// TwinCAT 3 PLC project PLC1
// Title: Projektnamn
// Company: Oaks AB
// ProgramVersion: 3.1.4023.0
// libraries:
//   OaksLibrary, * (OaksAB)
//   oaksModbusLibrary, * (Oaks AB)
//   Tc2_ModbusSrv, * (Beckhoff Automation GmbH)
//   Tc2_Standard, * (Beckhoff Automation GmbH)
//   Tc2_SUPS, * (Beckhoff Automation GmbH)
//   Tc2_System, * (Beckhoff Automation GmbH)
//   Tc2_Utilities, * (Beckhoff Automation GmbH)
//   Tc3_BA, * (Beckhoff Automation GmbH)
//   Tc3_Module, * (Beckhoff Automation GmbH)
// project tree:
//   GVLs/ IPadresser.TcGVL
//   / PlcTask.TcTTO
//   POUs/ImplicitChecks/ CheckBounds.TcPOU, CheckDivDInt.TcPOU, CheckDivLInt.TcPOU, CheckDivLReal.TcPOU, CheckDivReal.TcPOU, CheckLRangeSigned.TcPOU, CheckLRangeUnsigned.TcPOU, CheckRangeSigned.TcPOU, CheckRangeUnsigned.TcPOU
//   POUs/Lokala block/ fbDamperIndication_STL.TcPOU, fbfreezAlarm_markvarme.TcPOU, fbHeatPumpSr_StartStopDelay.TcPOU, fbReadAdsRealOutdoorMeantempWp_STL.TcPOU, fbTripleMotorControl_STL.TcPOU, fbTwinMotorControl_STL.TcPOU, fbTwinMotorHeatWoV.TcPOU
//   POUs/ MAIN.TcPOU
//   POUs/Övrigt/ AS101.TcPOU, KV1.TcPOU, S1.TcPOU, VVC1.TcPOU
// real-time tasks:
//   TASK PlcTask: cycle T#20ms, priority 20, ADS port 350
// I/O:
//   DEVICE Device 2 (CX-BK)
//     Box 1 (CX-BK)
// variable links:
//   PLC1/PLC1 Instance <-> Device 2 (CX-BK)/Box 1 (CX-BK)
//     PlcTask Inputs/AS101.AUT.V3 <-> Term 2 (KL1408)/Channel 6/Input
//     PlcTask Inputs/AS101.CBL.V3 <-> Term 2 (KL1408)/Channel 2/Input
//     PlcTask Inputs/AS101.FASBROTT.V3 <-> Term 2 (KL1408)/Channel 1/Input
//     PlcTask Inputs/AS101.JFB.V3 <-> Term 2 (KL1408)/Channel 4/Input
//     PlcTask Inputs/AS101.OSP.V3 <-> Term 2 (KL1408)/Channel 5/Input
//     PlcTask Inputs/AS101.RST.V <-> Term 2 (KL1408)/Channel 3/Input
//     PlcTask Inputs/AS101.SYSTEM.nKbusState <-> Inputs/State
//     PlcTask Inputs/KV1.PPA201_V <-> Term 5 (KL1408)/Channel 7/Input
//     PlcTask Inputs/S1.P11_QB_V3 <-> Term 2 (KL1408)/Channel 7/Input
//     PlcTask Inputs/S1.P12_QB_V3 <-> Term 4 (KL1408)/Channel 1/Input
//     PlcTask Inputs/S1.P13_QB_V3 <-> Term 4 (KL1408)/Channel 3/Input
//     PlcTask Inputs/S1.P14_QB_V3 <-> Term 4 (KL1408)/Channel 5/Input
//     PlcTask Inputs/S1.P15_QB_V3 <-> Term 4 (KL1408)/Channel 7/Input
//     PlcTask Inputs/S1.P16_QB_V3 <-> Term 5 (KL1408)/Channel 1/Input
//     PlcTask Inputs/S1.P17_QB_V3 <-> Term 5 (KL1408)/Channel 4/Input
//     PlcTask Inputs/S1.P11_V <-> Term 2 (KL1408)/Channel 8/Input
//     PlcTask Inputs/S1.P13_V <-> Term 4 (KL1408)/Channel 4/Input
//     PlcTask Inputs/S1.P15_V <-> Term 4 (KL1408)/Channel 8/Input
//     PlcTask Inputs/S1.P16_V <-> Term 5 (KL1408)/Channel 2/Input
//     PlcTask Inputs/S1.P17_V <-> Term 5 (KL1408)/Channel 5/Input
//     PlcTask Inputs/S1.P16_RC91_V <-> Term 5 (KL1408)/Channel 3/Input
//     PlcTask Inputs/S1.P17_RC91_V <-> Term 5 (KL1408)/Channel 6/Input
//     PlcTask Inputs/S1.ST1_P12_V <-> Term 4 (KL1408)/Channel 2/Input
//     PlcTask Inputs/S1.ST1_P14_V <-> Term 4 (KL1408)/Channel 6/Input
//     PlcTask Inputs/VVC1.GT420.iDataIn <-> Term 7 (KL3208-0010-4)/Channel 1/Data In
//     PlcTask Inputs/VVC1.GT420.usiState <-> Term 7 (KL3208-0010-4)/Channel 1/State
//     PlcTask Outputs/AS101.TCH1_bOutput <-> Term 3 (KL2809)/Channel 2/Output
//     PlcTask Outputs/AS101.TCH2_bOutput <-> Term 3 (KL2809)/Channel 3/Output
//     PlcTask Outputs/KV1.PPA201.CMD <-> Term 3 (KL2809)/Channel 11/Output
//     PlcTask Outputs/S1.P11.CMD <-> Term 3 (KL2809)/Channel 4/Output
//     PlcTask Outputs/S1.P13.CMD <-> Term 3 (KL2809)/Channel 6/Output
//     PlcTask Outputs/S1.P15.CMD <-> Term 3 (KL2809)/Channel 8/Output
//     PlcTask Outputs/S1.P16.CMD <-> Term 3 (KL2809)/Channel 9/Output
//     PlcTask Outputs/S1.P17.CMD <-> Term 3 (KL2809)/Channel 10/Output
//     PlcTask Outputs/S1.ST1_P12.CMD <-> Term 3 (KL2809)/Channel 5/Output
//     PlcTask Outputs/S1.ST1_P14.CMD <-> Term 3 (KL2809)/Channel 7/Output
//     PlcTask Outputs/VVC1.GT420.iDataOut <-> Term 7 (KL3208-0010-4)/Channel 1/Data Out
//     PlcTask Outputs/VVC1.GT420.usiCtrl <-> Term 7 (KL3208-0010-4)/Channel 1/Ctrl
//     PlcTask Outputs/oaksGVL.bSummalarm <-> Term 3 (KL2809)/Channel 1/Output

CONFIGURATION PLC1
    RESOURCE PLC ON TwinCAT3
        TASK PlcTask(INTERVAL := T#20ms, PRIORITY := 20);
        PROGRAM MAIN WITH PlcTask : MAIN;
    END_RESOURCE
END_CONFIGURATION

// ---- GVLs/IPadresser.TcGVL
{attribute 'qualified_only'}
VAR_GLOBAL PERSISTENT
	//Global lista för hantering av IP-adresser/portar i program. 
	//Vid ändring av IP-adress i drift kan man göra detta från webport-debugen. Välj enhet, datatyp STRING, adress IPadresser.sIPAddrElvaco1 (eller vad den i ditt fall heter). 
	//Tryck Läs för att se att den ip som förväntas läses in. Ändra till den nya önskade ip-adressen.
	
	//Glöm ej att ändra init-värdet här nedan så att vi sedan har koll på vilken ip-adress det ska vara i projektet!


	//sIPAddrElvaco1 : STRING := '192.168.1.31';

	//sIPAddrModbus1 : STRING := '192.168.1.41'; 
	//nTCPPortModbus1 : UINT := 502;
	
	//sIPAddrModbus2 : STRING := '192.168.1.42'; 
	//nTCPPortModbus2 : UINT := 5021;
	//nTCPPortModbus2 : UINT := 5022;
	//nTCPPortModbus2 : UINT := 5023;
	//nTCPPortModbus2 : UINT := 5024;
	
	//metz1_modbusTCP : ST_ModbusTCP := (sIPAddr:='192.168.0.111', nTCPPort:=502,iModbusLoop:=1);

	//amsNetId_AS11 : STRING :=	'5.97.77.211.1.1';
	///amsNetId_AS12 : STRING :=	'5.97.78.39.1.1';
	//amsNetId_AS31 : STRING :=	'5.97.78.42.1.1';
	//amsNetId_AS32 : STRING :=	'5.97.78.18.1.1';
	//amsNetId_AS34 : STRING :=	'5.97.78.33.1.1';
	//amsNetId_AS61 : STRING :=	'5.97.78.30.1.1';
	//amsNetId_AS62 : STRING :=	'5.97.77.235.1.1';
END_VAR

// ---- POUs/MAIN.TcPOU
PROGRAM MAIN
VAR
END_VAR

//Apparatskåp
AS101();
KV1();
S1();
VVC1();

END_PROGRAM

// ---- POUs/Övrigt/AS101.TcPOU
PROGRAM AS101
VAR
	PUMPMOTION: fbPumpMotion;
	WATCHDOG: fbWatchdogSwitching;
	RST: fbResetButton;
	CBL: fbFirealarm;
	AUT: fbFusealarm;
	JFB: fbJfb;
	OSP: fbOvervoltageProtection;
	MODBUS: fbModbusSekvensArray;
	SYSTEM: fbOaksSystem;
	TCH1: fbTimeChannelWp;
	TCH2: fbTimeChannelWp;
	ODT: fbReadAdsRealOutdoorMeantempWp_STL;	
	FASBROTT: fbDigitalAlarmIO;		
	ASTRO: fbSunClock := (SP1 := 57.7089, SP2 := 11.9746); 
	F_trigVentilmotion: F_TRIG;
	TOF_Ventilmotion: TOF;		

END_VAR
VAR_OUTPUT
	TCH1_bOutput AT %Q* : BOOL; //Tidkanal 1
	TCH2_bOutput AT %Q* : BOOL; //Tidkanal 2
	bVentilmotion: BOOL; //Ventilmotion aktiv~wp:[trendoptions]i:14400, t:1	
	FASBROTT_AL:BOOL; //larm fasbrottsrelä~wp:
	

END_VAR
VAR PERSISTENT

END_VAR

TCH2(); // fbTimeChannelWp
MODBUS(); // fbModbusSekvensArray
TCH1_bOutput := TCH1.bStart;
CBL(bInvert := true, bAutoReset := TRUE); // fbFirealarm
F_trigVentilmotion(CLK := PUMPMOTION.V); // F_TRIG
RST(); // fbResetButton
TCH2_bOutput := TCH2.bStart;
AUT(bInvert := false, bAutoReset := TRUE); // fbFusealarm
TCH1(); // fbTimeChannelWp
SYSTEM(); // fbOaksSystem
ODT(Enable := TRUE, AmsNetId := '111.111.11.1.1', sApparatskap := 'ASx', AdsPort := 851, AdsTimeout := T#60S); // fbReadAdsRealOutdoorMeantempWp_STL
PUMPMOTION(); // fbPumpMotion
FASBROTT(bInvert := TRUE, bAutoReset := TRUE); // fbDigitalAlarmIO
FASBROTT_AL := FASBROTT.bOutput;
WATCHDOG(); // fbWatchdogSwitching
JFB(bInvert := true, bAutoReset := TRUE); // fbJfb
OSP(bInvert := true, bAutoReset := TRUE); // fbOvervoltageProtection
TOF_Ventilmotion(IN := F_trigVentilmotion.Q); // TOF
bVentilmotion := TOF_Ventilmotion.Q;
// 		Göteborg SP1 = 57.7089 SP2 = 11.9746
// 		Stockholm SP1 = 59.3293 SP2 = 18.0686
// 		Malmö SP1 = 55.6050 SP2 = 13.0038
// 		Karlstad SP1 = 59.4022 SP2 = 13.5115
//
// 		För att hitta andra städers koordinater googla "Vilka koordinater har STAD?"
ASTRO(); // fbSunClock

END_PROGRAM

// ---- POUs/Lokala block/fbReadAdsRealOutdoorMeantempWp_STL.TcPOU
//Standard utetemperatur via ADS + handställning
FUNCTION_BLOCK fbReadAdsRealOutdoorMeantempWp_STL
VAR_INPUT
	Enable			: BOOL := TRUE;					// Start
	AmsNetId    	: T_AmsNetId; 					// AMS Net ID till enhet som skall avläsas
	sApparatskap 	: STRING 	:= 'ASXX'; 			// Skriv här vilket apparatskåp utetemperaturen tas emot från. Endast för visning i PV4-tagg.
    AdsPort     	: T_AmsPort := 851; 			// ADS-port till den enhet som skall avläsas
	AdsTimeout    	: TIME := DEFAULT_ADS_TIMEOUT; 	// ADS-timout
	Interval		: TIME := T#10S;				// Önskat intervall för läsning
	ErrDelay		: TIME := T#5S;					// Larmfördröjning för fel
	UseFallback		: BOOL;							// Sätts om fallbackvärde ska användas automatiskt vid fel
	FallbackVal		: REAL := 0.0;					// Värde vid kom.fel eller manuellt val av fallback (knyt t ex lokal utegivare om den finns)
	ForceFallback	: BOOL;							// Sätts om fallbackvärde ska användas ovillkorligt
END_VAR
VAR_OUTPUT
	{attribute 'OPC.UA.DA' := '1'}
	PV  AT %M* : REAL; //Utetemperatur hämtat från apparatskåp via ads.~wp:[unit]°C[format]0.0
	{attribute 'OPC.UA.DA' := '1'}
	PV1  AT %M* : REAL; //Utetemperatur medel hämtat från apparatskåp via ads.~wp:[unit]°C[format]0.0
	{attribute 'OPC.UA.DA' := '1'}
	FAULT AT %M* : BOOL; //Kommunikationsfel mottagning utetemperatur~wp:
	{attribute 'OPC.UA.DA' := '1'}
	PV4 AT %M* : STRING;   //Inställt amsNetId och apparatskåp~wp:
	AL8 AT %M* : BOOL; //Givare handställd~wp:[alarmoptions]p:3:
END_VAR
VAR	
	fbUtetempMom	: fbReadADSReal;
	fbUtetempMed	: fbReadADSReal;
	fbAlarm1: fbAlarm;
	
END_VAR
VAR_INPUT PERSISTENT
	OPM AT %M*: REAL;//Värde handställning~wp:[unit]%[format]0[trendoptions]i:14400, t:1
	M AT %M* : BOOL; //Handställning~wp:[trendoptions]i:14400, t:1
END_VAR

IF enable THEN
	fbUtetempMom(Enable := enable, amsNetId := amsNetId, adsPort := adsPort, adsTimeout := adsTimeout, symbolName := 'oaksGVL.rOutdoorTemp', interval := interval, errDelay := errDelay, fallbackVal := fallbackVal, useFallback := UseFallback, forceFallback := forceFallback);
	oaksGVL.rOutdoorTemp := SEL(M, fbUtetempMom.rOutputVar, OPM);
	
	fbUtetempMed(Enable := enable, amsNetId := amsNetId, adsPort := adsPort, adsTimeout := adsTimeout, symbolName := 'oaksGVL.rOutdoorTempMean', interval := interval, errDelay := errDelay, fallbackVal := fallbackVal, useFallback := UseFallback, forceFallback := forceFallback);
	oaksGVL.rOutdoorTempMean := fbUtetempMed.rOutputVar;
	
	PV		:= oaksGVL.rOutdoorTemp;							// Skriv utetemp till utvariabel	
	PV1		:= oaksGVL.rOutdoorTempMean;						// Skriv utetemp medel till utvariabel				
	PV4		:= CONCAT(amsNetId, CONCAT('-', sApparatskap));		// Bygg ihop ID-sträng för visning
	FAULT	:= fbUtetempMom.bErr OR fbUtetempMed.bErr;			// Sätt fel
	
	//Handställningslarm
	fbAlarm1(bInput:=M , tAlarmDelay:= , bAutoReset:=TRUE , bAlarmOutput=>AL8 );
END_IF;

END_FUNCTION_BLOCK

// ---- POUs/Övrigt/KV1.TcPOU
PROGRAM KV1
VAR
	PPA201_V AT %I*: BOOL; 	//Indikering~wp:[trendoptions]i:14400, t:1	
	PPA201: fbDigitalSignalLogic;
END_VAR

PPA201(
	bStart:= TRUE, 
	bSafe:= TRUE, 
	bHandsetBlock:= , 
	tStartDelay:= , 
	tStopDelay:= , 
	CMD=> , 
	AL8=> , 
	STATE1=> , 
	tStartDelayRemaining=> , 
	tStopDelayRemaining=> , 
	M:= , 
	MCMD:= );

END_PROGRAM

// ---- POUs/Övrigt/S1.TcPOU
PROGRAM S1
VAR
	larm1: fbalarm;
	larm2: fbalarm;
	larm3: fbalarm;
	larm4: fbalarm;
	larm5: fbalarm;
	larm6: fbalarm;
	larm7: fbalarm;	
END_VAR
VAR_OUTPUT
	P11_QB_AL: BOOL;	//Frånslagen säkerhetsbrytare~wp:[trendoption]i:300[alarmoptions]p:B	
	P12_QB_AL: BOOL;	//Frånslagen säkerhetsbrytare~wp:[trendoption]i:300[alarmoptions]p:B	
	P13_QB_AL: BOOL;	//Frånslagen säkerhetsbrytare~wp:[trendoption]i:300[alarmoptions]p:B	
	P14_QB_AL: BOOL;	//Frånslagen säkerhetsbrytare~wp:[trendoption]i:300[alarmoptions]p:B	
	P15_QB_AL: BOOL;	//Frånslagen säkerhetsbrytare~wp:[trendoption]i:300[alarmoptions]p:B		
	P16_QB_AL: BOOL;	//Frånslagen säkerhetsbrytare~wp:[trendoption]i:300[alarmoptions]p:B
	P17_QB_AL: BOOL;	//Frånslagen säkerhetsbrytare~wp:[trendoption]i:300[alarmoptions]p:B	
	P11: fbDigitalSignalLogic;	
	ST1_P12: fbDigitalSignalLogic;
	P13: fbDigitalSignalLogic;
	ST1_P14: fbDigitalSignalLogic;
	P15: fbDigitalSignalLogic;	
	P16: fbDigitalSignalLogic;
	P17: fbDigitalSignalLogic;	
END_VAR
VAR_INPUT
	P11_QB_V3 AT %I*: BOOL; 	//Larmingång~wp:[trendoptions]i:14400, t:1	
	P12_QB_V3 AT %I*: BOOL; 	//Larmingång~wp:[trendoptions]i:14400, t:1
	P13_QB_V3 AT %I*: BOOL; 	//Larmingång~wp:[trendoptions]i:14400, t:1
	P14_QB_V3 AT %I*: BOOL; 	//Larmingång~wp:[trendoptions]i:14400, t:1
	P15_QB_V3 AT %I*: BOOL; 	//Larmingång~wp:[trendoptions]i:14400, t:1	
	P16_QB_V3 AT %I*: BOOL; 	//Larmingång~wp:[trendoptions]i:14400, t:1
	P17_QB_V3 AT %I*: BOOL; 	//Larmingång~wp:[trendoptions]i:14400, t:1	
	
	
	P11_V AT %I*: BOOL; 	//Indikering~wp:[trendoptions]i:14400, t:1	
	ST1_P12_V AT %I*: BOOL; 	//Indikering~wp:[trendoptions]i:14400, t:1
	P13_V AT %I*: BOOL; 	//Indikering~wp:[trendoptions]i:14400, t:1
	ST1_P14_V AT %I*: BOOL; 	//Indikering~wp:[trendoptions]i:14400, t:1
	P15_V AT %I*: BOOL; 	//Indikering~wp:[trendoptions]i:14400, t:1	
	P16_V AT %I*: BOOL; 	//Indikering~wp:[trendoptions]i:14400, t:1
	P17_V AT %I*: BOOL; 	//Indikering~wp:[trendoptions]i:14400, t:1	


	P16_RC91_V AT %I*: BOOL; 	//Indikering hög nivå~wp:[trendoptions]i:14400, t:1	
	P17_RC91_V AT %I*: BOOL; 	//Indikering hög nivå~wp:[trendoptions]i:14400, t:1		
END_VAR

P11(bStart:= TRUE, 	bSafe:= NOT AS101.CBL.AL, 	bHandsetBlock:= , 	tStartDelay:= , 	tStopDelay:= , 	CMD=> , 	AL8=> , 	STATE1=> , 	tStartDelayRemaining=> , 	tStopDelayRemaining=> , 	M:= , 	MCMD:= );
ST1_P12(bStart:= TRUE, 	bSafe:= NOT AS101.CBL.AL, 	bHandsetBlock:= , 	tStartDelay:= , 	tStopDelay:= , 	CMD=> , 	AL8=> , 	STATE1=> , 	tStartDelayRemaining=> , 	tStopDelayRemaining=> , 	M:= , 	MCMD:= );
P13(	bStart:= TRUE, 	bSafe:= NOT AS101.CBL.AL, 	bHandsetBlock:= , 	tStartDelay:= , 	tStopDelay:= , 	CMD=> , 	AL8=> , 	STATE1=> , 	tStartDelayRemaining=> , 	tStopDelayRemaining=> , 	M:= , 	MCMD:= );
ST1_P14(bStart:= TRUE, 	bSafe:= NOT AS101.CBL.AL, 	bHandsetBlock:= , 	tStartDelay:= , 	tStopDelay:= , 	CMD=> , 	AL8=> , 	STATE1=> , 	tStartDelayRemaining=> , 	tStopDelayRemaining=> , 	M:= , 	MCMD:= );
P15(	bStart:= TRUE, 	bSafe:= NOT AS101.CBL.AL, 	bHandsetBlock:= , 	tStartDelay:= , 	tStopDelay:= , 	CMD=> , 	AL8=> , 	STATE1=> , 	tStartDelayRemaining=> , 	tStopDelayRemaining=> , 	M:= , 	MCMD:= );
P16(	bStart:= TRUE, 	bSafe:= NOT AS101.CBL.AL, 	bHandsetBlock:= , 	tStartDelay:= , 	tStopDelay:= , 	CMD=> , 	AL8=> , 	STATE1=> , 	tStartDelayRemaining=> , 	tStopDelayRemaining=> , 	M:= , 	MCMD:= );
P17(	bStart:= TRUE, 	bSafe:= NOT AS101.CBL.AL, 	bHandsetBlock:= , 	tStartDelay:= , 	tStopDelay:= , 	CMD=> , 	AL8=> , 	STATE1=> , 	tStartDelayRemaining=> , 	tStopDelayRemaining=> , 	M:= , 	MCMD:= );

//larm
larm6(bInput:= NOT P11_QB_V3, tAlarmDelay:= T#3S, bAutoReset:= TRUE, bAlarmOutput=> P11_QB_AL);
larm1(bInput:= NOT P12_QB_V3, tAlarmDelay:= T#3S, bAutoReset:= TRUE, bAlarmOutput=> P12_QB_AL);
larm2(bInput:= NOT P13_QB_V3, tAlarmDelay:= T#3S, bAutoReset:= TRUE, bAlarmOutput=> P13_QB_AL);
larm3(bInput:= NOT P14_QB_V3, tAlarmDelay:= T#3S, bAutoReset:= TRUE, bAlarmOutput=> P14_QB_AL);
larm4(bInput:= NOT P15_QB_V3, tAlarmDelay:= T#3S, bAutoReset:= TRUE, bAlarmOutput=> P15_QB_AL);
larm5(bInput:= NOT P16_QB_V3, tAlarmDelay:= T#3S, bAutoReset:= TRUE, bAlarmOutput=> P16_QB_AL);
larm7(bInput:= NOT P17_QB_V3, tAlarmDelay:= T#3S, bAutoReset:= TRUE, bAlarmOutput=> P17_QB_AL);

END_PROGRAM

// ---- POUs/Övrigt/VVC1.TcPOU
PROGRAM VVC1
VAR
	GT420: fbPT1000;
	larm1: fbLowLimitAlarm;
END_VAR
VAR PERSISTENT
	GT420_LAD: REAL := 30; //Larmfördröjning låg temperatur~wp:[unit]min
	GT420_ALL: REAL := 45; //Larmgräns låg temperatur~wp:[unit]°C[format]0.0[trendoption]i:300
END_VAR
VAR_OUTPUT
	GT420_LAL	: BOOL; //Larm låg VVC returtemp~wp:[alarmoptions]p:C
END_VAR

GT420(
	M:= , 
	iSensorType:= , 
	iTerminalType:= , 
	bPt100:= , 
	bFaultVal:= , 
	rFaultVal:= , 
	PV=> , 
	FAULT=> , 
	AL8=> , 
	OPM:= , 
	rCal:= , 
	iMedelvardeSekunder:= );
	
larm1(	bInput:= ,	tAlarmDelay:= fRealToMinute(GT420_LAD),	bAutoReset:= TRUE,	bAlarmOutput=> GT420_LAL,	bEnable:= TRUE,	rProcessValue:= GT420.PV,rLowLimit:= GT420_ALL);

END_PROGRAM

// ---- POUs/ImplicitChecks/CheckBounds.TcPOU
FUNCTION CheckBounds : DINT
VAR_INPUT
	index, lower, upper: DINT;
END_VAR

{noflow}

IF  index < lower THEN
	CheckBounds := lower;
	oaksGVL.udiCheckBounds := oaksGVL.udiCheckBounds + 1;
ELSIF  index > upper THEN
	CheckBounds := upper;
	oaksGVL.udiCheckBounds := oaksGVL.udiCheckBounds + 1;
ELSE  
	CheckBounds := index;
END_IF
{flow}

END_FUNCTION

// ---- POUs/ImplicitChecks/CheckDivDInt.TcPOU
FUNCTION CheckDivDInt : DINT
VAR_INPUT
	divisor:DINT;
END_VAR

{noflow}
IF divisor = 0 THEN
	CheckDivDInt:=1;
	oaksGVL.udiCheckDivDInt := oaksGVL.udiCheckDivDInt + 1;
ELSE
	CheckDivDInt:=divisor;
END_IF;
{flow}

END_FUNCTION

// ---- POUs/ImplicitChecks/CheckDivLInt.TcPOU
FUNCTION CheckDivLInt : LINT
VAR_INPUT
	divisor:LINT;
END_VAR

{noflow}
IF divisor = 0 THEN
	CheckDivLInt:=1;
	oaksGVL.udiCheckDivLInt := oaksGVL.udiCheckDivLInt + 1;	
ELSE
	CheckDivLInt:=divisor;
END_IF;
{flow}

END_FUNCTION

// ---- POUs/ImplicitChecks/CheckDivLReal.TcPOU
FUNCTION CheckDivLReal : LREAL
VAR_INPUT
	divisor:LREAL;
END_VAR

{noflow}
IF divisor = 0 THEN
	CheckDivLReal:=1;
	oaksGVL.udiCheckDivLReal := oaksGVL.udiCheckDivLReal + 1;
ELSE
	CheckDivLReal:=divisor;
END_IF;
{flow}

END_FUNCTION

// ---- POUs/ImplicitChecks/CheckDivReal.TcPOU
FUNCTION CheckDivReal : REAL
VAR_INPUT
	divisor:REAL;
END_VAR

{noflow}
IF divisor = 0 THEN
	oaksGVL.udiCheckDivReal := oaksGVL.udiCheckDivReal + 1;
	CheckDivReal := 1;
ELSE
	CheckDivReal:=divisor;
END_IF;
{flow}

END_FUNCTION

// ---- POUs/ImplicitChecks/CheckLRangeSigned.TcPOU
FUNCTION CheckLRangeSigned : LINT
VAR_INPUT
	value, lower, upper: LINT;
END_VAR

{noflow}

IF (value < lower) THEN
	CheckLRangeSigned := lower;
	oaksGVL.udiCheckLRangeSigned := oaksGVL.udiCheckLRangeSigned + 1;
ELSIF(value > upper) THEN
	CheckLRangeSigned := upper;
	oaksGVL.udiCheckLRangeSigned := oaksGVL.udiCheckLRangeSigned + 1;
ELSE
	CheckLRangeSigned := value;
END_IF

{flow}

END_FUNCTION

// ---- POUs/ImplicitChecks/CheckLRangeUnsigned.TcPOU
FUNCTION CheckLRangeUnsigned : ULINT
VAR_INPUT
	value, lower, upper: ULINT;
END_VAR

{noflow}

IF (value < lower) THEN
	CheckLRangeUnsigned := lower;
	oaksGVL.udiCheckLRangeUnsigned := oaksGVL.udiCheckLRangeUnsigned + 1;
ELSIF(value > upper) THEN
	CheckLRangeUnsigned := upper;
	oaksGVL.udiCheckLRangeUnsigned := oaksGVL.udiCheckLRangeUnsigned + 1;
ELSE
	CheckLRangeUnsigned := value;
END_IF
{flow}

END_FUNCTION

// ---- POUs/ImplicitChecks/CheckRangeSigned.TcPOU
FUNCTION CheckRangeSigned : DINT
VAR_INPUT
	value, lower, upper: DINT;
END_VAR

{noflow}

IF (value < lower) THEN
	CheckRangeSigned := lower;
	oaksGVL.udiCheckRangeSigned := oaksGVL.udiCheckRangeSigned + 1;
ELSIF(value > upper) THEN
	CheckRangeSigned := upper;
	oaksGVL.udiCheckRangeSigned := oaksGVL.udiCheckRangeSigned + 1;
ELSE
	CheckRangeSigned := value;
END_IF
{flow}

END_FUNCTION

// ---- POUs/ImplicitChecks/CheckRangeUnsigned.TcPOU
FUNCTION CheckRangeUnsigned : UDINT
VAR_INPUT
	value, lower, upper: UDINT;
END_VAR

{noflow}

IF (value < lower) THEN
	CheckRangeUnsigned := lower;
	oaksGVL.udiCheckRangeUnsigned := oaksGVL.udiCheckRangeUnsigned + 1;
ELSIF(value > upper) THEN
	CheckRangeUnsigned := upper;
	oaksGVL.udiCheckRangeUnsigned := oaksGVL.udiCheckRangeUnsigned + 1;
ELSE
	CheckRangeUnsigned := value;
END_IF
{flow}

END_FUNCTION

// ---- POUs/Lokala block/fbDamperIndication_STL.TcPOU
FUNCTION_BLOCK fbDamperIndication_STL
VAR_INPUT
	bStart : BOOL; // startvillkor
	bSafe: BOOL; // Säkerhetsvillkor
	bHandsetBlock : BOOL; // Används för blockering av handställning utan att blockera utsignal i autoläge. OBS! - För säkerhetsvillkor se ingång bSafe!
	tStartDelay : TIME := T#0S; // Startfördröjning
	tStopDelay : TIME := T#0S; // Stoppfördröjning
	tAlarmDelay : TIME := T#180S; // Larmfördröjning
END_VAR
VAR_OUTPUT
	{attribute 'OPC.UA.DA' := '1'}
	CMD AT %Q* : BOOL; //Utsignal~wp:[trendoptions]i:14400, t:1
	{attribute 'OPC.UA.DA' := '1'}
	AL8 AT %M* : BOOL; //Utsignal handställd~wp:[alarmoptions]p:3
	{attribute 'OPC.UA.DA' := '1'}
	V0 AT %I* : BOOL; //Stängtindikering~wp:[trendoptions]i:14400, t:1
	{attribute 'OPC.UA.DA' := '1'}
	V1 AT %I* : BOOL; //Öppetindikering~wp:[trendoptions]i:14400, t:1
	{attribute 'OPC.UA.DA' := '1'}
	AL AT %M* : BOOL; //Spjällfel~wp:
	STATE1 AT %M* : STRING; //Status IO-modul~wp:
	tStartDelayRemaining : TIME; // Aktuell  återstående tid startfördröjning
	tStopDelayRemaining : TIME; // Aktuell återstående tid toppfördröjning
END_VAR
VAR
	bInternalStart : BOOL;
	fbAlarm2 : fbAlarm; // Larm handställning
	//Handställningsvariabler från IO
	TI_bStateAuto AT %I* :BOOL :=TRUE; //Status Auto/Manuell
	TI_bStateRelay AT %I* :BOOL :=FALSE; //Status reläutgång
	bIOManual : BOOL;
	
	fbStartDelay: TON; // Startfördröjning
	fbStopDelay: TOF; // Stoppfördröjning
	
	fbAlarm1: fbAlarm;
	bAlarm: BOOL;
END_VAR
VAR_INPUT PERSISTENT
	{attribute 'OPC.UA.DA' := '1'}
	M AT %M* : BOOL; //Handställning~wp:[trendoptions]i:14400, t:1
	{attribute 'OPC.UA.DA' := '1'}
	MCMD AT %M* : BOOL; //Styrsignal handställning~wp:[trendoptions]i:14400, t:1
END_VAR

	//Handställning
	fbAlarm2(bInput:=M OR NOT TI_bStateAuto, tAlarmDelay:= , bAutoReset:=TRUE , bAlarmOutput=>AL8 );
	
	IF NOT bSafe OR bHandsetBlock THEN
		M := FALSE;
	END_IF;
	
	//Manuell omkopplare IO-modul
	bIOManual := fKx2652State(bAuto := TI_bStateAuto, bRelayStatus := TI_bStateRelay, sState => STATE1);
	
	
	//Start-/stoppfördröjning
    fbStartDelay(IN:=bStart , PT:=tStartDelay , Q=> , ET=> );
	fbStopDelay(IN:=fbStartDelay.Q, PT:=tStopDelay , Q=> , ET=> );
	
	tStopDelayRemaining:= (fbStopDelay.PT - fbStopDelay.ET);
	tStartDelayRemaining:=(fbStartDelay.PT - fbStartDelay.ET);
	
	bInternalStart := fbStopDelay.Q;
	
	IF NOT TI_bStateAuto THEN
		CMD := bIOManual;
	ELSE
		CMD := (((bInternalStart AND NOT M) OR (M AND MCMD)) AND bSafe) OR bIOManual;
	END_IF
	
	//Larm
	bAlarm := (NOT CMD AND NOT V0) OR (CMD AND NOT V1);

	fbAlarm1(bInput:=bAlarm , tAlarmDelay:=tAlarmDelay , bAutoReset:= TRUE, bAlarmOutput=> AL);

END_FUNCTION_BLOCK

// ---- POUs/Lokala block/fbfreezAlarm_markvarme.TcPOU
FUNCTION_BLOCK fbfreezAlarm_markvarme EXTENDS fbFreezeAlarm
//Frysvaktsblock med integrerad handställbar pt1000-givare. Handställning förreglas om insignal underskrider 12 grader eller vid givarfel.
//Minbegränsning returtemperatur vid drift stopp aggregat går ej att ställa under 10°C.

VAR_INPUT
	bOperationIndication : BOOL; // Driftindikering för tilluftsfläkt kopplas hit. Används för att avgöra vilket minbegränsningsbörvärde som skall användas.
END_VAR
VAR_OUTPUT
	{attribute 'OPC.UA.DA' := '1'}
	LAL AT %M* : BOOL; //Frysvakt~wp:[alarmoptions]p:1,rst:OAKSGVL_RST=1
	rMinOutput : REAL; // Utsignal minbegränsning returvattenregulator 
END_VAR
VAR
	fbReg01 : Tc3_BA_Common.FB_BA_PIDCtrl;
	rSetpoint : REAL;
	fbFreezeInterlock : fbAlarm;
	//itemp :INT;
	{attribute 'OPC.UA.DA' := '1'}
	PV8 AT %M* : REAL; //Aktuell reglersignal minbegränsningsregulator~wp:[unit]%[format]0[trendoptions]i:300
END_VAR
VAR_INPUT PERSISTENT
	{attribute 'OPC.UA.DA' := '1'}
	ALL AT %M* : REAL := 7; //Larmgräns frysvakt~wp:[unit]°C[format]0.0
	{attribute 'OPC.UA.DA' := '1'}
	SP1 AT %M* : REAL := 12; //Minbegränsning returtemperatur vid drift av pump~wp:[unit]°C[format]0.0
	{attribute 'OPC.UA.DA' := '1'}
	SP2 AT %M* : REAL := 15; //Minbegränsning returtemperatur vid drift stopp av pump~wp:[unit]°C[format]0.0
END_VAR

	SUPER^();

	//Handställning förreglas om insignal underskrider 12 grader eller vid givarfel
	IF FB_BA_AI01.rVal < 12 OR FAULT THEN
		M := FALSE;
	END_IF
	
	// Minbegränsning av frysvaktsinställning 5 grader
	IF ALL < 5.0 THEN 
		ALL := 5.0;
	END_IF

	
	// Frysvaktslarm om temperatur underskrider inställt värde. 
	fbFreezeInterlock(
	bInput:= PV < ALL OR FAULT, 
	tAlarmDelay:= T#3S , 
	bAutoReset:=FALSE , 
	bAlarmOutput=> LAL);
	
	
	// Minbegränsning av inställningsvärde för returtemperatur vid stopp av aggregat
	IF SP2 < 10.0 THEN 
		SP2 := 10.0;
	END_IF
	// Val av börvärde till minbegränsningsregulator
	IF bOperationIndication THEN
		rSetpoint := SP1;
	ELSE
		rSetpoint := SP2;
	END_IF
	
	fbReg01(
	bEn:=TRUE , 
	rW:=rSetpoint , 
	rX:=PV , 
	udiOpMode:= , 
	bActn:= , 
	rKp:= 20, 
	udiTn_ms:= , 
	udiTv_ms:= , 
	udiTd_ms:= , 
	rYMax:=100 , 
	rYMin:= 0, 
	rNZ:= , 
	udiCycCl:= , 
	bSync:= , 
	rSync:= , 
	rY=> , 
	rE=> , 
	bARW=> );
	
	IF NOT FAULT THEN
		rMinOutput := fbReg01.rY;
	ELSE
		rMinOutput := 100;
	END_IF
	// För visning och trendning i webport
	PV8 := rMinOutput;

END_FUNCTION_BLOCK

// ---- POUs/Lokala block/fbHeatPumpSr_StartStopDelay.TcPOU
// Block för start/stopp på utetemperatur. Utgången går till då utetemp underskrider inställt värde under inställd tid 
// eller när utetemp underskrider gräns för direktstart. Utgången går från då utetemperatur överstigit inställt värde under inställd tid.
FUNCTION_BLOCK fbHeatPumpSr_StartStopDelay
VAR_INPUT
	rOutdoorTemp : ANY; // Utetemperatur Knyter man inget här används oaksGVL.rOutdoortemp
END_VAR
VAR_IN_OUT 
	rDirectStart	: REAL; // Starta bOutput utan fördröjning då rOutdoorTemp underskrider
	rStartLimit 	: REAL; // Starta bOutput då rOutdoorTemp underskrider
	rStopLimit 		: REAL; // Stoppa bOutput då rOutdoorTemp överstiger
	iStopDelay 		: INT;  // Stoppfördröjning
	iStartDelay		: INT;  // Startfördröjning

END_VAR
VAR_OUTPUT
	bOutput 		: BOOL; // Utsignal
	bStopDelayOdt 	: BOOL; // Stoppfördröjning aktiv via utetemperatur
	bStartDelayOdt 	: BOOL; // Startfördröjning aktiv via utetemperatur
END_VAR
VAR
	rTempUsed 		: REAL; // Uteluftstemperatur
	bInternalStart 	: BOOL;
	fbPumpTof : TOF;
	fbPumpTon : TON;
END_VAR

//Temp select
	rTempUsed := F_GetTempToUse(rOutdoorTemp);

IF  rStartLimit > rStopLimit THEN
	rStopLimit := rStartLimit + 1;
END_IF

IF rTempUsed < rStartLimit  THEN
	bInternalStart := TRUE;
ELSIF rTempUsed > rStopLimit THEN
	bInternalStart := FALSE;	
END_IF

fbPumpTon(IN:=bInternalStart , PT:=INT_TO_TIME(iStartDelay)*60000 , Q=> , ET=> );
fbPumpTof(IN:=fbPumpTon.Q OR (rTempUsed < MAX(rDirectStart, 5.0)) , PT:=INT_TO_TIME(iStopDelay)*60000  , Q=> , ET=> );

//Startfördröjning aktiv
bStartDelayOdt :=  bInternalStart AND NOT fbPumpTon.Q;
//Stoppfördröjning aktiv
bStopDelayOdt := NOT bInternalStart AND fbPumpTof.Q;


bOutput:= fbPumpTof.Q ;

END_FUNCTION_BLOCK

// ---- POUs/Lokala block/fbTripleMotorControl_STL.TcPOU
FUNCTION_BLOCK fbTripleMotorControl_STL
VAR_INPUT
	{attribute 'OPC.UA.DA' := '1'}
	bStart AT %M* : BOOL; //Startvilkor
	bError1,bError2,bError3 : BOOL;
	{attribute 'OPC.UA.DA' := '1'}
	M AT %M*  : BOOL; //Manuell pumpväxling~wp:

	rAnalogInput1 : REAL; //Analog ingång för steg 1
	rAnalogInput2 : REAL; //Analog ingång för steg 2
	rStartDelaySupportPump: REAL; //Startfördröjning paralleldrift
	rStopDelaySupportPump: REAL; //Stoppfördröjning paralleldrift
END_VAR
VAR_OUTPUT
	{attribute 'OPC.UA.DA' := '1'}
	PV AT %M* : INT; //Aktuellt pumpval~wp:[trendoption]i:300
	bStartOutput1,bStartOutput2, bStartOutput3 : BOOL;
	{attribute 'OPC.UA.DA' := '1'}
	AL AT %M* : BOOL; //Driftfel trillingpumpar~wp:[trendoption]i:300[alarmoptions]p:1:
	rAnalogOutput1, rAnalogOutput2, rAnalogOutput3: REAL; //Utsignal till motorer
	bSupportPumpActive: BOOL; //Paralleldrift aktiv
END_VAR
VAR 
	fbDayTrig: R_trig;
	
	
	nActualDayCase	: INT;
	nActualHour 	: INT;
	nActualMinute 	: INT;
	
	nTime : INT; // Internvariabel aktuell tid (nActualHour+nActualMinute)
	
	bDay : BOOL; // Internvariabel blir TRUE om inställd dag är lika med aktuell dag
	bTime : BOOL; // Internvariabel blir TRUE om inställd tid är lika med aktuell tid

	fbHandsetToN: TON;
	
	
	fbAlarm1 : fbAlarm;
	
	
	fbChangeTON1 : TON;
	fbChangeTOF1 : TOF;
	
	bStartSupportPump: BOOL;
END_VAR
VAR_INPUT PERSISTENT
	{attribute 'OPC.UA.DA' := '1'}
	SP1 AT %M*  : INT:=1; //Dag för pumpväxling (-1 = ingen växling 0 = Söndag 1 = Måndag 2 = Tisdag..6 = Söndag~wp:
	{attribute 'OPC.UA.DA' := '1'}
	SP2 AT %M*  : INT:=1000; //Tid för pumpväxling~wp:[format]00:00[engmin]0[engmax]2400
END_VAR


	fbHandsetToN.PT := T#1S;
	fbHandsetToN(IN:=M);
	
	IF fbHandsetToN.Q THEN 
		M := FALSE;
	END_IF

	nActualDayCase := oaksGVL.iDayOfWeek;
	nActualHour := oaksGVL.iHour*100;
	nActualMinute :=oaksGVL.iMinute;
	
	// nActualHour+nActualMinute
	
	nTime := nActualHour+nActualMinute;
	
	bDay := nActualDayCase = SP1;
	bTime := nTime = SP2;


	IF SP1 < -1 OR  SP1>7 THEN
		SP1 := 1;
	END_IF
	
	IF SP2 < 0 OR  SP2>2359 THEN
		SP2 := 1200;
	END_IF

	IF PV < 1 OR PV > 3  THEN	
		PV := 1;
	END_IF;
	
	IF (bDay AND bTime) OR M THEN
		fbDayTrig(CLK := TRUE);
	ELSE
		fbDayTrig(CLK := FALSE);
	END_IF

	IF fbDayTrig.Q THEN
		IF PV = 1 THEN
			PV := 2;
		ELSIF PV = 2 THEN
			PV:= 3;
		ELSE
			PV := 1;
		END_IF
	END_IF
	
	IF rAnalogInput1 = 100 THEN
		bStartSupportPump:= TRUE;
	ELSE 
		bStartSupportPump:= FALSE;
	END_IF
	
	
	fbChangeTON1(IN:= bStartSupportPump, PT:= fRealToMinute(rStartDelaySupportPump), Q=> , ET=> );
	fbChangeTOF1(IN:= fbChangeTON1.Q, PT:= fRealToMinute(rStopDelaySupportPump), Q=> , ET=> );
	
	bStartOutput1 := (((PV = 1 OR PV = 3) AND NOT bError1) OR (bError2 OR bError3)) AND bStart OR (bStart AND fbChangeTOF1.Q);
	bStartOutput2 := (((PV = 1 OR PV = 2) AND NOT bError2) OR (bError1 OR bError3)) AND bStart OR (bStart AND fbChangeTOF1.Q);
	bStartOutput3 := (((PV = 2 OR PV = 3) AND NOT bError3) OR (bError2 OR bError1)) AND bStart OR (bStart AND fbChangeTOF1.Q);

	
//Analog utsignal, vid larmande primärpump körs reservpump enligt sekvens 1.
	IF PV = 1 THEN
			IF NOT (bError1 OR bError2) THEN
				rAnalogOutput1:= rAnalogInput1 ;
				rAnalogOutput2:= rAnalogInput1 ;
				rAnalogOutput3:= rAnalogInput2 ;
			ELSIF  bError1 OR bError2 THEN
				rAnalogOutput1:= rAnalogInput1 ;
				rAnalogOutput2:= rAnalogInput1 ;
				rAnalogOutput3:= rAnalogInput1 ;
			END_IF
		ELSIF PV = 2 THEN
			IF NOT (bError2 OR bError3) THEN
				rAnalogOutput1:= rAnalogInput2 ;
				rAnalogOutput2:= rAnalogInput1 ;
				rAnalogOutput3:= rAnalogInput1 ;
			ELSIF bError2 OR bError3 THEN
				rAnalogOutput1:= rAnalogInput1 ;
				rAnalogOutput2:= rAnalogInput1 ;
				rAnalogOutput3:= rAnalogInput1 ;
			END_IF
		ELSIF PV = 3 THEN
			IF NOT (bError1 OR bError3) THEN
				rAnalogOutput1:= rAnalogInput1 ;
				rAnalogOutput2:= rAnalogInput2 ;
				rAnalogOutput3:= rAnalogInput1 ;
			ELSIF bError1 OR bError3 THEN
				rAnalogOutput1:= rAnalogInput1 ;
				rAnalogOutput2:= rAnalogInput1 ;
				rAnalogOutput3:= rAnalogInput1 ;
			END_IF
		END_IF
	
	
//Larm
	bSupportPumpActive:= bStart AND fbChangeTOF1.Q;
	fbAlarm1(bInput:= bError1 AND bError2 AND bError3, tAlarmDelay:= T#3S , bAutoReset:=TRUE , bAlarmOutput=> AL);

END_FUNCTION_BLOCK

// ---- POUs/Lokala block/fbTwinMotorControl_STL.TcPOU
FUNCTION_BLOCK fbTwinMotorControl_STL
VAR_INPUT
	{attribute 'OPC.UA.DA' := '1'}
	bStart AT %M* : BOOL; //Startvilkor
	bError1,bError2 : BOOL;
	{attribute 'OPC.UA.DA' := '1'}
	M AT %M*  : BOOL; //Manuell pumpväxling~wp:

	rAnalogInput1 : REAL; //Analog ingång för steg 1
	rStartDelaySupportPump: REAL; //Startfördröjning paralleldrift
	rStopDelaySupportPump: REAL; //Stoppfördröjning paralleldrift
END_VAR
VAR_OUTPUT
	{attribute 'OPC.UA.DA' := '1'}
	PV AT %M* : INT; //Aktuellt pumpval~wp:[trendoption]i:300
	bStartOutput1,bStartOutput2 : BOOL;
	{attribute 'OPC.UA.DA' := '1'}
	AL AT %M* : BOOL; //Driftfel parpumpar~wp:[trendoption]i:300[alarmoptions]p:1
	bSupportPumpActive: BOOL; //Paralleldrift aktiv
END_VAR
VAR 
	fbDayTrig: R_trig;
	
	
	nActualDayCase	: INT;
	nActualHour 	: INT;
	nActualMinute 	: INT;
	
	nTime : INT; // Internvariabel aktuell tid (nActualHour+nActualMinute)
	
	bDay : BOOL; // Internvariabel blir TRUE om inställd dag är lika med aktuell dag
	bTime : BOOL; // Internvariabel blir TRUE om inställd tid är lika med aktuell tid

	fbHandsetToN: TON;
	
	
	fbAlarm1 : fbAlarm;
	
	
	fbChangeTON1 : TON;
	fbChangeTOF1 : TOF;
	
	bStartSupportPump: BOOL;
END_VAR
VAR_INPUT PERSISTENT
	{attribute 'OPC.UA.DA' := '1'}
	SP1 AT %M*  : INT:=1; //Dag för pumpväxling (-1 = ingen växling 0 = Söndag 1 = Måndag 2 = Tisdag..6 = Söndag~wp:
	{attribute 'OPC.UA.DA' := '1'}
	SP2 AT %M*  : INT:=1000; //Tid för pumpväxling~wp:[format]00:00[engmin]0[engmax]2400
END_VAR


	fbHandsetToN.PT := T#1S;
	fbHandsetToN(IN:=M);
	
	IF fbHandsetToN.Q THEN 
		M := FALSE;
	END_IF

	nActualDayCase := oaksGVL.iDayOfWeek;
	nActualHour := oaksGVL.iHour*100;
	nActualMinute :=oaksGVL.iMinute;
	
	// nActualHour+nActualMinute
	
	nTime := nActualHour+nActualMinute;
	
	bDay := nActualDayCase = SP1;
	bTime := nTime = SP2;


	IF SP1 < -1 OR  SP1>7 THEN
		SP1 := 1;
	END_IF
	
	IF SP2 < 0 OR  SP2>2359 THEN
		SP2 := 1200;
	END_IF

	IF PV < 1 OR PV > 2  THEN	
		PV := 1;
	END_IF;
	
	IF (bDay AND bTime) OR M THEN
		fbDayTrig(CLK := TRUE);
	ELSE
		fbDayTrig(CLK := FALSE);
	END_IF

	IF fbDayTrig.Q THEN
		IF PV = 1 THEN
			PV := 2;
		ELSE
			PV := 1;
		END_IF
	END_IF
	
	IF rAnalogInput1 = 100 THEN
		bStartSupportPump:= TRUE;
	ELSE 
		bStartSupportPump:= FALSE;
	END_IF
	
	
	fbChangeTON1(IN:= bStartSupportPump, PT:= fRealToMinute(rStartDelaySupportPump), Q=> , ET=> );
	fbChangeTOF1(IN:= fbChangeTON1.Q, PT:= fRealToMinute(rStopDelaySupportPump), Q=> , ET=> );
	
	bStartOutput1 := ((PV = 1 AND NOT bError1) OR bError2) AND bStart OR (bStart AND fbChangeTOF1.Q);
	bStartOutput2 := ((PV = 2 AND NOT bError2) OR bError1) AND bStart OR (bStart AND fbChangeTOF1.Q);

	bSupportPumpActive:= bStart AND fbChangeTOF1.Q;
	
	fbAlarm1(bInput:= bError1 AND bError2 , tAlarmDelay:= T#3S , bAutoReset:=TRUE , bAlarmOutput=> AL);

END_FUNCTION_BLOCK

// ---- POUs/Lokala block/fbTwinMotorHeatWoV.TcPOU
FUNCTION_BLOCK fbTwinMotorHeatWoV
VAR_INPUT
	{attribute 'OPC.UA.DA' := '1'}
	V AT %M* : BOOL; //Startsignal~wp:[trendoption]i:300
	bError1,bError2 : BOOL;
	{attribute 'OPC.UA.DA' := '1'}
	M AT %M*  : BOOL; //Manuell pumpväxling~wp:
	rOutdoorTemp : ANY; //Utetemperatur används för start/stopp Knyter man inget här används oaksGVL.rOutdoortemp
	bCustomStartCon : BOOL := TRUE; //Om ytterligare villkor för start/stopp finns lägg detta här
	
	rAnalogInput1 : REAL; //Analog ingång för steg 1
	rAnalogInput2 : REAL; //Analog ingång för steg 2
END_VAR
VAR_OUTPUT
	{attribute 'OPC.UA.DA' := '1'}
	PV AT %M* : INT; //Aktuellt pumpval~wp:[trendoption]i:300
	bStartOutput1,bStartOutput2 : BOOL;
	{attribute 'OPC.UA.DA' := '1'}
	AL AT %M* : BOOL; //Driftfel parpumpar~wp:[trendoption]i:300[alarmoptions]p:1:
END_VAR
VAR 
	fbDayTrig: R_trig;
	
	
	nActualDayCase	: INT;
	nActualHour 	: INT;
	nActualMinute 	: INT;
	
	nTime : INT; // Internvariabel aktuell tid (nActualHour+nActualMinute)
	
	bDay : BOOL; // Internvariabel blir TRUE om inställd dag är lika med aktuell dag
	bTime : BOOL; // Internvariabel blir TRUE om inställd tid är lika med aktuell tid

	fbHandsetToN: TON;
	
	
	fbAlarm1 : fbAlarm;
	
	fbHeatPumpSr1 : fbHeatPumpSr;
	rTempUsed : REAL; //Uteluftstemperatur
	
	fbChangeTON1, fbChangeTON2 : TON;
	fbChangeTOF1, fbChangeTOF2 : TOF;
	
	bStartSupport1, bStartSupport2 : BOOL;
END_VAR
VAR_INPUT PERSISTENT
	{attribute 'OPC.UA.DA' := '1'}
	SP1 AT %M*  : INT:=1; //Dag för pumpväxling (-1 = ingen växling 0 = Söndag 1 = Måndag 2 = Tisdag..6 = Söndag~wp:
	{attribute 'OPC.UA.DA' := '1'}
	SP2 AT %M*  : INT:=1000; //Tid för pumpväxling~wp:[format]00:00[engmin]0[engmax]2400
	{attribute 'OPC.UA.DA' := '1'}
	SP7 AT %M* : INT := 15; //Stoppfördröjning~wp:[unit]min
	{attribute 'OPC.UA.DA' := '1'}
	SP3 AT %M* : REAL := 17;  //Stoppa värmesystem om utetemp överstiger~wp:[unit]°C[format]0.0
	{attribute 'OPC.UA.DA' := '1'}
	SP4 AT %M* : REAL := 14; //Starta värmesystem om utetemp underskrider~wp:[unit]°C[format]0.0
	
	{attribute 'OPC.UA.DA' := '1'}
	SP5 AT %M*  : REAL:=10; //Starta stödpump då utsignal är 100% i~wp:[unit]min[format]0
	{attribute 'OPC.UA.DA' := '1'}
	SP6 AT %M*  : REAL:=5; //Stoppa stödpump då utsignal är 0% i~wp:[unit]min[format]0
END_VAR

//Temp select
	rTempUsed := F_GetTempToUse(rOutdoorTemp);
	
fbHeatPumpSr1(
	rOutdoorTemp:=rTempUsed , 
	rStartLimit:= SP4, 
	rStopLimit:=SP3 , 
	iStopDelay:=SP7 , 
	bOutput=> );
	
	V := fbHeatPumpSr1.bOutput AND bCustomStartCon;

	fbHandsetToN.PT := T#1S;
	fbHandsetToN(IN:=M);
	
	IF fbHandsetToN.Q THEN 
		M := FALSE;
	END_IF

	nActualDayCase := oaksGVL.iDayOfWeek;
	nActualHour := oaksGVL.iHour*100;
	nActualMinute :=oaksGVL.iMinute;
	
	// nActualHour+nActualMinute
	
	nTime := nActualHour+nActualMinute;
	
	bDay := nActualDayCase = SP1;
	bTime := nTime = SP2;


	IF SP1 < -1 OR  SP1>7 THEN
		SP1 := 1;
	END_IF
	
	IF SP2 < 0 OR  SP2>2359 THEN
		SP2 := 1200;
	END_IF

	IF PV < 1 OR PV > 2  THEN	
		PV := 1;
	END_IF;
	
	IF (bDay AND bTime) OR M THEN
		fbDayTrig(CLK := TRUE);
	ELSE
		fbDayTrig(CLK := FALSE);
	END_IF

	IF fbDayTrig.Q THEN
		IF PV = 1 THEN
			PV := 2;
		ELSE
			PV := 1;
		END_IF
	END_IF
	
	IF (PV = 1) AND (rAnalogInput1 = 100) THEN
		bStartSupport2 := TRUE;
	ELSIF (PV = 1) (* AND (rAnalogInput2 = 0) *) AND (rAnalogInput1 < 100) THEN
		bStartSupport2 := FALSE;
	END_IF
	
	fbChangeTON1(IN:= bStartSupport2, PT:= fRealToMinute(rMinute:= SP5), Q=> , ET=> );
	fbChangeTOF1(IN:= fbChangeTON1.Q, PT:= fRealToMinute(rMinute:= SP6), Q=> , ET=> );
	
	IF (PV = 2) AND (rAnalogInput2 = 100) THEN
		bStartSupport1 := TRUE;
	ELSIF (PV = 2) (* AND (rAnalogInput1 = 0) *) AND (rAnalogInput2 < 100) THEN
		bStartSupport1 := FALSE;
	END_IF
	
	fbChangeTON2(IN:= bStartSupport1, PT:= fRealToMinute(rMinute:= SP5), Q=> , ET=> );
	fbChangeTOF2(IN:= fbChangeTON2.Q, PT:= fRealToMinute(rMinute:= SP6), Q=> , ET=> );
	
	bStartOutput1 := (((PV = 1 AND NOT bError1) OR bError2) OR fbChangeTOF2.Q) AND V ;
	bStartOutput2 := (((PV = 2 AND NOT bError2) OR bError1) OR fbChangeTOF1.Q) AND V;

	fbAlarm1(bInput:= bError1 AND bError2 , tAlarmDelay:= T#3S , bAutoReset:=TRUE , bAlarmOutput=> AL);

END_FUNCTION_BLOCK
